(* IEC 61131-3 sources: repolevel_ST_code_completion/output/full_case_fixed/repoeval_PT1Filter/readful_result_history, 4 files *)

(* ---- FB_PT1Filter_0.st ---- *)
FUNCTION_BLOCK FB_PT1Filter
VAR_INPUT
	rInput: REAL:= 0.0; 								//输入数据
	rK: REAL:= 1.0; 									//增益
	tT: TIME; 											//时间参数
END_VAR
VAR_OUTPUT
	rOutput: REAL:= 0.0;  								//输出数据
END_VAR
VAR
	_rT: LREAL;
	_rY: LREAL;
END_VAR

_rT := TIME_TO_REAL(tT) / 10.0;  // Convert time constant to real and adjust for sampling period

IF _rT = 0.0 THEN
	rOutput := rInput;  // Initialize output if time constant is zero
ELSIF ABS(rOutput - rInput) < 1E-6 THEN
	rOutput := rInput;  // Prevent division by zero
ELSIF _rT > 0.0 THEN
	rOutput := (rK / _rT) * rInput + (1.0 - (1.0 / _rT)) * _rY;  // Apply PT1 filter formula
ELSE
	rOutput := rInput;  // If time constant is less than or equal to zero, output equals input
END_IF

_rY := rOutput;  // Update internal state
END_FUNCTION_BLOCK

(* ---- FB_PT1Filter_1.st ---- *)
FUNCTION_BLOCK FB_PT1Filter
VAR_INPUT
	rInput: REAL:= 0.0; 								//输入数据
	rK: REAL:= 1.0; 									//增益
	tT: TIME; 											//时间参数
END_VAR
VAR_OUTPUT
	rOutput: REAL:= 0.0;  								//输出数据
END_VAR
VAR
	_rT: LREAL;
	_rY: LREAL;
END_VAR

// Replace TIME_TO_REAL(tT) with direct TIME-to-real scaling
_rT := REAL_TO_LREAL(TO_REAL(tT / T#1ms) / 10.0);  // Convert time constant (TIME) to real for sampling

IF _rT = 0.0 THEN
	rOutput := rInput;  // Initialize output if time constant is zero
ELSIF ABS(rOutput - rInput) < 1E-6 THEN
	rOutput := rInput;  // Prevent division by zero
ELSIF _rT > 0.0 THEN
// Protect against division-by-zero scenarios where _rT <= 1E-6
rOutput := (rT > 1E-6) AND (rK / _rT) * rInput + (1.0 - (1.0 / _rT)) * _rY ELSE rInput;
ELSE
	rOutput := rInput;  // If time constant is less than or equal to zero, output equals input
END_IF

_rY := rOutput;  // Update internal state
END_FUNCTION_BLOCK

(* ---- FB_PT1Filter_2.st ---- *)
FUNCTION_BLOCK FB_PT1Filter
VAR_INPUT
	rInput: REAL:= 0.0; 								//输入数据
	rK: REAL:= 1.0; 									//增益
	tT: TIME; 											//时间参数
END_VAR
VAR_OUTPUT
	rOutput: REAL:= 0.0;  								//输出数据
END_VAR
VAR
	_rT: LREAL;
	_rY: LREAL;
END_VAR

// Replace TIME_TO_REAL(tT) with direct TIME-to-real scaling
_rT := REAL_TO_LREAL(TO_REAL(tT / T#1ms) / 10.0);  // Convert time constant (TIME) to real for sampling

IF _rT = 0.0 THEN
	rOutput := rInput;  // Initialize output if time constant is zero
ELSIF ABS(rOutput - rInput) < 1E-6 THEN
	rOutput := rInput;  // Prevent division by zero
ELSIF _rT > 0.0 THEN
// Correct syntax and replace rT with _rT
IF (_rT > 1E-6) THEN
  rOutput := (rK / _rT) * rInput + (1.0 - (1.0 / _rT)) * _rY;  // Apply PT1 filter formula
ELSE
  rOutput := rInput;  // Output equals input for invalid _rT
END_IF;
ELSE
	rOutput := rInput;  // If time constant is less than or equal to zero, output equals input
END_IF

_rY := rOutput;  // Update internal state
END_FUNCTION_BLOCK

(* ---- FB_PT1Filter_3.st ---- *)
FUNCTION_BLOCK FB_PT1Filter
VAR_INPUT
	rInput: REAL:= 0.0; 								//输入数据
	rK: REAL:= 1.0; 									//增益
	tT: TIME; 											//时间参数
END_VAR
VAR_OUTPUT
	rOutput: REAL:= 0.0;  								//输出数据
END_VAR
VAR
	_rT: LREAL;
	_rY: LREAL;
END_VAR

// Replace TIME_TO_REAL(tT) with direct TIME-to-real scaling
_rT := REAL_TO_LREAL(TO_REAL(tT / T#1ms) / 10.0);  // Convert time constant (TIME) to real for sampling

IF _rT = 0.0 THEN
	rOutput := rInput;  // Initialize output if time constant is zero
ELSIF ABS(rOutput - rInput) < 1E-6 THEN
	rOutput := rInput;  // Prevent division by zero
ELSIF _rT > 0.0 THEN
// Simplify the conditional logic and handle _rT cases appropriately
IF (_rT > 1E-6) THEN
  rOutput := (rK / _rT) * rInput + (1.0 - (1.0 / _rT)) * _rY;  // Apply PT1 filter formula
ELSE
  rOutput := rInput;  // Output equals input for invalid or small _rT
END_IF;
ELSE
	rOutput := rInput;  // If time constant is less than or equal to zero, output equals input
END_IF

_rY := rOutput;  // Update internal state
END_FUNCTION_BLOCK
